{attribute 'qualified_only'}
//{attribute 'strict'}
{attribute 'to_string'}
TYPE E_LogicIfConditionOperator :
(
	GRT := 0,
	LES := 1,
	EQU := 2,
	GRE := 3,
	LEQ := 4
);
END_TYPE

(* stored: Version 1.1.0.1
   EnumerationTextList E_LogicIfConditionOperator: Id {c9313150-3151-42c0-916a-cfda4a20649d} *)
